FUNCTION_BLOCK SDODatenMotor1
VAR_INPUT
END_VAR
VAR_OUTPUT
	
	Motor1Spannung: UINT;
	Motor1Strom: INT;
	Motor1Strombegrenzung: UINT;
	Motor1Regelfehler: INT;
	Motor1Geschwindigkeit: INT;
	Motor1Overloadtime: UINT;
	Motor1Overtemperature: BOOL;
	Motor1Torqueoverload: BOOL;
	Motor1Shortcirciut: BOOL;
	
END_VAR
VAR
	Motorspannung: FB_EcCoESdoRead;	
	Motorstrom: FB_EcCoESdoRead;
	Strombegrenzung: FB_EcCoESdoRead;
	Regelfehler: FB_EcCoESdoRead;
	Geschwindigkeit: FB_EcCoESdoRead;
	Overload: FB_EcCoESdoRead;
	Short_Circuit: FB_EcCoESdoRead;
	Torque_Overload: FB_EcCoESdoRead;
	Over_Temperature: FB_EcCoESdoRead;

	trigger: BOOL;
	TON_0: TON;
	TON_1: TON;
	ms: TIME;

END_VAR

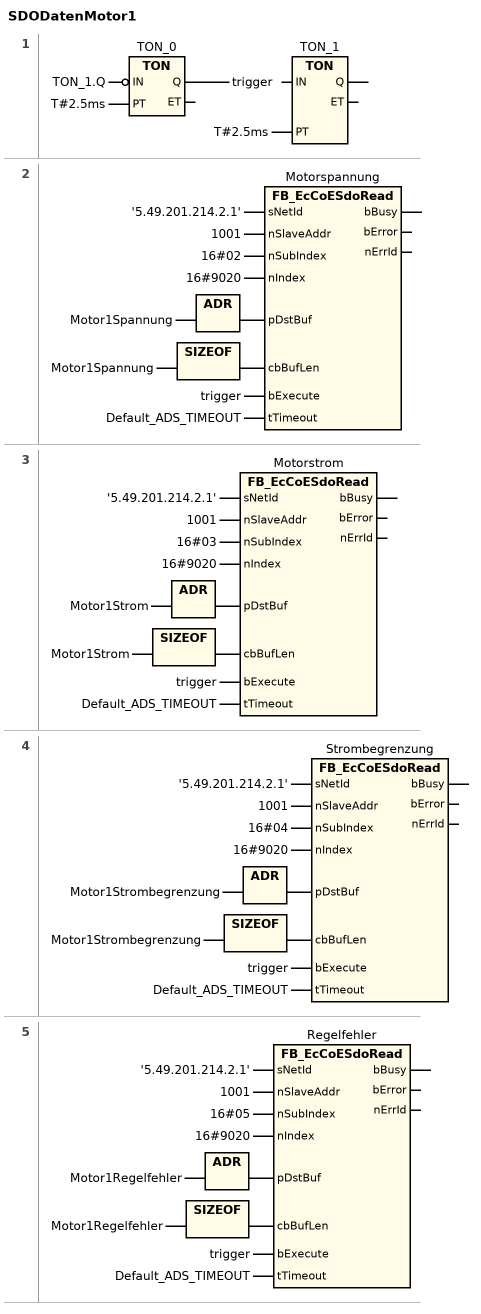
// NETWORK 1
TON_0(IN := NOT TON_1.Q, PT := T#2.5ms); // TON
trigger := TON_0.Q;
TON_1(IN := TON_0.Q, PT := T#2.5ms); // TON

// NETWORK 2
Motorspannung(
    sNetId := '5.49.201.214.2.1',
    nSlaveAddr := 1001,
    nSubIndex := 16#02,
    nIndex := 16#9020,
    pDstBuf := ADR(Motor1Spannung),
    cbBufLen := SIZEOF(Motor1Spannung),
    bExecute := trigger,
    tTimeout := Default_ADS_TIMEOUT); // FB_EcCoESdoRead

// NETWORK 3
Motorstrom(
    sNetId := '5.49.201.214.2.1',
    nSlaveAddr := 1001,
    nSubIndex := 16#03,
    nIndex := 16#9020,
    pDstBuf := ADR(Motor1Strom),
    cbBufLen := SIZEOF(Motor1Strom),
    bExecute := trigger,
    tTimeout := Default_ADS_TIMEOUT); // FB_EcCoESdoRead

// NETWORK 4
Strombegrenzung(
    sNetId := '5.49.201.214.2.1',
    nSlaveAddr := 1001,
    nSubIndex := 16#04,
    nIndex := 16#9020,
    pDstBuf := ADR(Motor1Strombegrenzung),
    cbBufLen := SIZEOF(Motor1Strombegrenzung),
    bExecute := trigger,
    tTimeout := Default_ADS_TIMEOUT); // FB_EcCoESdoRead

// NETWORK 5
Regelfehler(
    sNetId := '5.49.201.214.2.1',
    nSlaveAddr := 1001,
    nSubIndex := 16#05,
    nIndex := 16#9020,
    pDstBuf := ADR(Motor1Regelfehler),
    cbBufLen := SIZEOF(Motor1Regelfehler),
    bExecute := trigger,
    tTimeout := Default_ADS_TIMEOUT); // FB_EcCoESdoRead

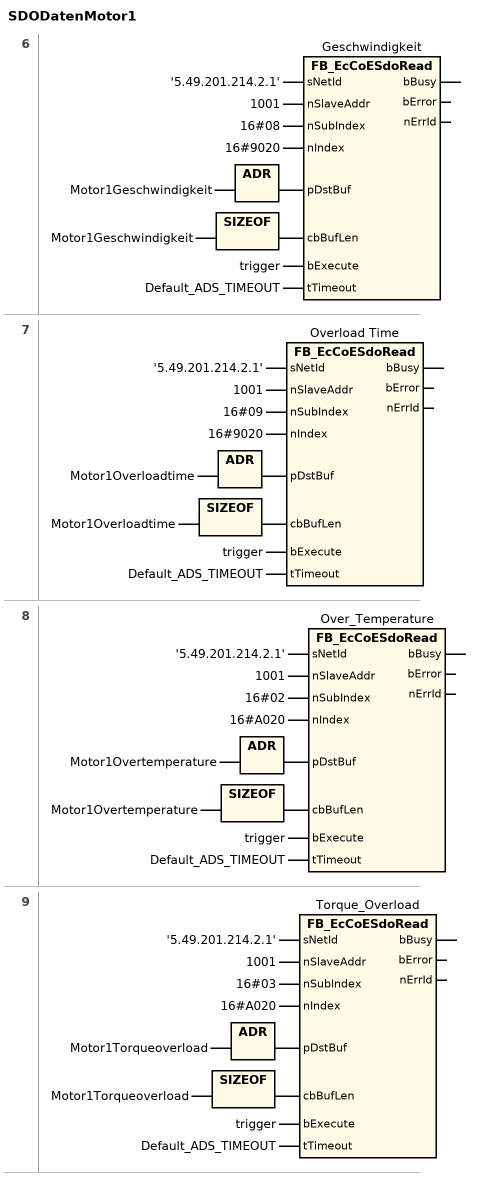
// NETWORK 6
Geschwindigkeit(
    sNetId := '5.49.201.214.2.1',
    nSlaveAddr := 1001,
    nSubIndex := 16#08,
    nIndex := 16#9020,
    pDstBuf := ADR(Motor1Geschwindigkeit),
    cbBufLen := SIZEOF(Motor1Geschwindigkeit),
    bExecute := trigger,
    tTimeout := Default_ADS_TIMEOUT); // FB_EcCoESdoRead

// NETWORK 7
Overload Time(
    sNetId := '5.49.201.214.2.1',
    nSlaveAddr := 1001,
    nSubIndex := 16#09,
    nIndex := 16#9020,
    pDstBuf := ADR(Motor1Overloadtime),
    cbBufLen := SIZEOF(Motor1Overloadtime),
    bExecute := trigger,
    tTimeout := Default_ADS_TIMEOUT); // FB_EcCoESdoRead

// NETWORK 8
Over_Temperature(
    sNetId := '5.49.201.214.2.1',
    nSlaveAddr := 1001,
    nSubIndex := 16#02,
    nIndex := 16#A020,
    pDstBuf := ADR(Motor1Overtemperature),
    cbBufLen := SIZEOF(Motor1Overtemperature),
    bExecute := trigger,
    tTimeout := Default_ADS_TIMEOUT); // FB_EcCoESdoRead

// NETWORK 9
Torque_Overload(
    sNetId := '5.49.201.214.2.1',
    nSlaveAddr := 1001,
    nSubIndex := 16#03,
    nIndex := 16#A020,
    pDstBuf := ADR(Motor1Torqueoverload),
    cbBufLen := SIZEOF(Motor1Torqueoverload),
    bExecute := trigger,
    tTimeout := Default_ADS_TIMEOUT); // FB_EcCoESdoRead

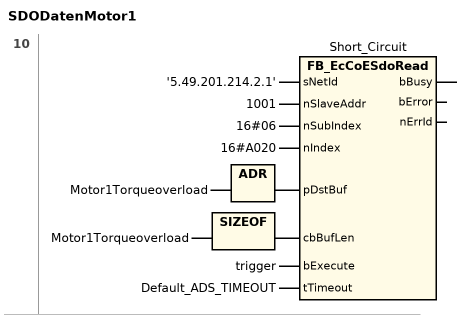
// NETWORK 10
Short_Circuit(
    sNetId := '5.49.201.214.2.1',
    nSlaveAddr := 1001,
    nSubIndex := 16#06,
    nIndex := 16#A020,
    pDstBuf := ADR(Motor1Torqueoverload),
    cbBufLen := SIZEOF(Motor1Torqueoverload),
    bExecute := trigger,
    tTimeout := Default_ADS_TIMEOUT); // FB_EcCoESdoRead

END_FUNCTION_BLOCK

(* stored: Version 1.1.0.1, ProductVersion 3.1.4020.12
   POU SDODatenMotor1: Id {db92f199-2295-40f9-97d2-319ddc0272f8}, SpecialFunc None *)
